// TIA Portal V20 export
DATA_BLOCK "BK12"   // DB291
// stored: MemoryReserve 100
   VAR
      "X10-1.ANODE NG P&P 1st BACKWARD" : Bool := FALSE;
      "X11-1.SPARE" : Bool := FALSE;
      "X12-1.ANODE NG P&P 2nd BACKWARD" : Bool := FALSE;
      "X13-1.SPARE" : Bool := FALSE;
      "X14-1.ANODE NG P&P UP" : Bool := TRUE;
      "X15-1.SPARE" : Bool := FALSE;
      "X16-1.ANODE NG P&P VACUUM PRESSURE SWITCH" : Bool := FALSE;
      "X17-1.SPARE" : Bool := FALSE;
      "X10-2.ANODE NG P&P 1st FORWARD" : Bool := FALSE;
      "X11-2.SPARE" : Bool := FALSE;
      "X12-2.ANODE NG P&P 2nd FORWARD" : Bool := FALSE;
      "X13-2.SPARE" : Bool := FALSE;
      "X14-2.ANODE NG P&P DOWN" : Bool := FALSE;
      "X15-2.SPARE" : Bool := FALSE;
      "X16-2.ANODE NG P&P ELECTRODE DETECT SENSOR" : Bool := TRUE;
      "X17-2.SPARE" : Bool := FALSE;
   END_VAR
BEGIN
END_DATA_BLOCK
